// STOP só funciona em MANUAL
IF M1a_ModeScada = 1 THEN
    M1a_stop := FALSE;
ELSIF M1a_ModeScada = 2 THEN
    GVL.Out[75] := GVL.Out[75] AND (NOT M1a_stop);
ELSE
	GVL.Out[75] := FALSE;
END_IF;

IF M1b_ModeScada = 1 THEN
    M1b_stop := FALSE;
ELSIF M1b_ModeScada = 2 THEN
    //GVL.Out[87] := GVL.Out[87] AND (NOT M1b_stop);
ELSE
	GVL.Out[87] := FALSE;
END_IF;

IF M1c_ModeScada = 1 THEN
    M1c_stop := FALSE;
ELSIF M1c_ModeScada = 2 THEN
    GVL.Out[99] := GVL.Out[99] AND (NOT M1c_stop);
ELSE
	GVL.Out[99] := FALSE;
END_IF;

// ======================================================
// BLOQUEAR CONVEYORS EM MANUAL ATÉ FINISH OPERATION
// ======================================================
GVL.Out[71] := GVL.Out[71] AND (NOT M1a_ConvHold); // conveyor M1a
//GVL.Out[83] := GVL.Out[83] AND (NOT M1b_ConvHold); // conveyor M1b
GVL.Out[95] := GVL.Out[95] AND (NOT M1c_ConvHold); // conveyor M1c

// ======================================================
// CHANGE TOOL M1a - CELL1 - MACHINE 1
// ======================================================

M1a_TargetTool := WORD_TO_INT(M1a_Tool_SCADA);
M1a_CurrentTool := INT_TO_WORD(M1a_CurrentToolID);
GVL.Out[73] := FALSE; // Rotate -
GVL.Out[74] := FALSE; // Rotate +

CASE M1a_ToolState OF
    0: // IDLE
        M1a_ToolSensorReady := FALSE;
        IF M1a_ChangeTool AND ((M1a_ModeScada = 2) OR (M1a_ModeScada = 3)) THEN
                IF M1a_TargetTool = M1a_CurrentToolID THEN
					M1a_ChangeTool := FALSE;
                    M1a_ToolState := 0;
                ELSE
                    M1a_ToolState := 10;
                END_IF;
        END_IF;
    10: // ROTATE
        // Tool 1
        IF M1a_CurrentToolID = 1 THEN
            IF M1a_TargetTool = 2 THEN
                GVL.Out[73] := TRUE; // Rotate -
            ELSIF M1a_TargetTool = 3 THEN
                GVL.Out[74] := TRUE; // Rotate +
            END_IF;
        // Tool 2
        ELSIF M1a_CurrentToolID = 2 THEN
            IF M1a_TargetTool = 3 THEN
                GVL.Out[73] := TRUE; // Rotate -
            ELSIF M1a_TargetTool = 1 THEN
                GVL.Out[74] := TRUE; // Rotate +
            END_IF;
        // Tool 3
        ELSIF M1a_CurrentToolID = 3 THEN
            IF M1a_TargetTool = 1 THEN
                GVL.Out[73] := TRUE; // Rotate -
            ELSIF M1a_TargetTool = 2 THEN
                GVL.Out[74] := TRUE; // Rotate +
            END_IF;
        END_IF;
        // Sensor da tool M1a
        IF NOT GVL.In[31] THEN
            M1a_ToolSensorReady := TRUE;
            M1a_ToolState := 20;
        END_IF;


    20: // CONTINUAR A RODAR ATÉ O SENSOR VOLTAR
        IF M1a_CurrentToolID = 1 THEN
            IF M1a_TargetTool = 2 THEN
                GVL.Out[73] := TRUE;
            ELSIF M1a_TargetTool = 3 THEN
                GVL.Out[74] := TRUE;
            END_IF;
        ELSIF M1a_CurrentToolID = 2 THEN
            IF M1a_TargetTool = 3 THEN
                GVL.Out[73] := TRUE;
            ELSIF M1a_TargetTool = 1 THEN
                GVL.Out[74] := TRUE;
            END_IF;
        ELSIF M1a_CurrentToolID = 3 THEN
            IF M1a_TargetTool = 1 THEN
                GVL.Out[73] := TRUE;
            ELSIF M1a_TargetTool = 2 THEN
                GVL.Out[74] := TRUE;
            END_IF;
        END_IF;
		
        IF M1a_ToolSensorReady AND GVL.In[31] THEN
            // Atualiza a tool interna da máquina
			M1a_CurrentToolID := M1a_TargetTool;
    		M1a_CurrentTool := INT_TO_WORD(M1a_CurrentToolID);
            GVL.Out[73] := FALSE;
            GVL.Out[74] := FALSE;
            M1a_ToolSensorReady := FALSE;
			M1a_ChangeTool := FALSE;
            M1a_ToolState := 0;
        END_IF;
END_CASE;

// ======================================================
// CHANGE TOOL M1b - CELL1 - MACHINE 2
// ======================================================

M1b_TargetTool := WORD_TO_INT(M1b_Tool_SCADA);
M1b_CurrentTool := INT_TO_WORD(M1b_CurrentToolID);
GVL.Out[85] := FALSE; // Rotate -
GVL.Out[86] := FALSE; // Rotate +

CASE M1b_ToolState OF
    0: // IDLE
        M1b_ToolSensorReady := FALSE;
        IF M1b_ChangeTool AND ((M1b_ModeScada = 2) OR (M1b_ModeScada = 3)) THEN
            IF M1b_TargetTool = M1b_CurrentToolID THEN
                M1b_ToolState := 0;
				M1b_ChangeTool := FALSE;
            ELSE
                M1b_ToolState := 10;
            END_IF;
        END_IF;

    10: // ROTATE
        // Tool 1
        IF M1b_CurrentToolID = 1 THEN
            IF M1b_TargetTool = 2 THEN
                GVL.Out[85] := TRUE; // Rotate -
            ELSIF M1b_TargetTool = 3 THEN
                GVL.Out[86] := TRUE; // Rotate +
            END_IF;
        // Tool 2
        ELSIF M1b_CurrentToolID = 2 THEN
            IF M1b_TargetTool = 3 THEN
                GVL.Out[85] := TRUE; // Rotate -
            ELSIF M1b_TargetTool = 1 THEN
                GVL.Out[86] := TRUE; // Rotate +
            END_IF;
        // Tool 3
        ELSIF M1b_CurrentToolID = 3 THEN
            IF M1b_TargetTool = 1 THEN
                GVL.Out[85] := TRUE; // Rotate -
            ELSIF M1b_TargetTool = 2 THEN
                GVL.Out[86] := TRUE; // Rotate +
            END_IF;
        END_IF;
        // Sensor da tool M1b
        IF NOT GVL.In[38] THEN
            M1b_ToolSensorReady := TRUE;
            M1b_ToolState := 20;
        END_IF;

    20: // CONTINUAR A RODAR ATÉ O SENSOR VOLTAR
        IF M1b_CurrentToolID = 1 THEN
            IF M1b_TargetTool = 2 THEN
                GVL.Out[85] := TRUE;
            ELSIF M1b_TargetTool = 3 THEN
                GVL.Out[86] := TRUE;
            END_IF;
        ELSIF M1b_CurrentToolID = 2 THEN
            IF M1b_TargetTool = 3 THEN
                GVL.Out[85] := TRUE;
            ELSIF M1b_TargetTool = 1 THEN
                GVL.Out[86] := TRUE;
            END_IF;
        ELSIF M1b_CurrentToolID = 3 THEN
            IF M1b_TargetTool = 1 THEN
                GVL.Out[85] := TRUE;
            ELSIF M1b_TargetTool = 2 THEN
                GVL.Out[86] := TRUE;
            END_IF;
        END_IF;
		
        IF M1b_ToolSensorReady AND GVL.In[38] THEN
            M1b_CurrentToolID := M1b_TargetTool;
            M1b_CurrentTool := INT_TO_WORD(M1b_CurrentToolID);
            GVL.Out[85] := FALSE;
            GVL.Out[86] := FALSE;
            M1b_ToolSensorReady := FALSE;
			M1b_ChangeTool := FALSE;
            M1b_ToolState := 0;
        END_IF;
END_CASE;

// ======================================================
// CHANGE TOOL M1c - CELL1 - MACHINE 3
// ======================================================

M1c_TargetTool := WORD_TO_INT(M1c_Tool_SCADA);
M1c_CurrentTool := INT_TO_WORD(M1c_CurrentToolID);
GVL.Out[97] := FALSE; // Rotate -
GVL.Out[98] := FALSE; // Rotate +

CASE M1c_ToolState OF
    0: // IDLE
        M1c_ToolSensorReady := FALSE;
        IF M1c_ChangeTool AND ((M1c_ModeScada = 2) OR (M1c_ModeScada = 3)) THEN
            IF M1c_TargetTool = M1c_CurrentToolID THEN
                M1c_ToolState := 0;
				M1c_ChangeTool := FALSE;
            ELSE
                M1c_ToolState := 10;
            END_IF;
        END_IF;

    10: // ROTATE
        // Tool 1
        IF M1c_CurrentToolID = 8 THEN
            IF M1c_TargetTool = 9 THEN
                GVL.Out[97] := TRUE; // Rotate -
            ELSIF M1c_TargetTool = 11 THEN
                GVL.Out[98] := TRUE; // Rotate +
            END_IF;
        // Tool 2
        ELSIF M1c_CurrentToolID = 9 THEN
            IF M1c_TargetTool = 11 THEN
                GVL.Out[97] := TRUE; // Rotate -
            ELSIF M1c_TargetTool = 8 THEN
                GVL.Out[98] := TRUE; // Rotate +
            END_IF;
        // Tool 3
        ELSIF M1c_CurrentToolID = 11 THEN
            IF M1c_TargetTool = 8 THEN
                GVL.Out[97] := TRUE; // Rotate -
            ELSIF M1c_TargetTool = 9 THEN
                GVL.Out[98] := TRUE; // Rotate +
            END_IF;
        END_IF;
		
        // Sensor da tool M1c
        IF NOT GVL.In[45] THEN
            M1c_ToolSensorReady := TRUE;
            M1c_ToolState := 20;
        END_IF;
		
    20: // CONTINUAR A RODAR ATÉ O SENSOR VOLTAR
        IF M1c_CurrentToolID = 8 THEN
            IF M1c_TargetTool = 9 THEN
                GVL.Out[97] := TRUE;
            ELSIF M1c_TargetTool = 11 THEN
                GVL.Out[98] := TRUE;
            END_IF;
        ELSIF M1c_CurrentToolID = 9 THEN
            IF M1c_TargetTool = 11 THEN
                GVL.Out[97] := TRUE;
            ELSIF M1c_TargetTool = 8 THEN
                GVL.Out[98] := TRUE;
            END_IF;
        ELSIF M1c_CurrentToolID = 11 THEN
            IF M1c_TargetTool = 8 THEN
                GVL.Out[97] := TRUE;
            ELSIF M1c_TargetTool = 9 THEN
                GVL.Out[98] := TRUE;
            END_IF;
        END_IF;

        IF M1c_ToolSensorReady AND GVL.In[45] THEN
            M1c_CurrentToolID := M1c_TargetTool;
            M1c_CurrentTool := INT_TO_WORD(M1c_CurrentToolID);
            GVL.Out[97] := FALSE;
            GVL.Out[98] := FALSE;
            M1c_ToolSensorReady := FALSE;
			M1c_ChangeTool := FALSE;
            M1c_ToolState := 0;
        END_IF;
END_CASE;

Gate0 := GVL.Out[71];
Gate1 := GVL.Out[81];
Gate2 := GVL.Out[83];
Gate3 := GVL.Out[93];
Gate4 := GVL.Out[95];
Gate5 := GVL.Out[75];
Gate6 := GVL.Out[87];
Gate7 := GVL.Out[99];
Gate8 := GVL.Out[29];
Gate9 := GVL.Out[49];
S_sensor1 := GVL.In[30];
S_sensor2 := GVL.In[36];
S_sensor3 := GVL.In[37];
S_sensor4 := GVL.In[43];
S_sensor5 := GVL.In[44];
S_sensor6 := GVL.In[11];
S_sensor7 := GVL.In[21];

END_PROGRAM
